TYPE EL5112_Data :
STRUCT
	{attribute addProperty Name "ENC Status Channel 1"}
	ENC_StatusChannel_1 : EL5112_ENC_StatusChannel;
	{attribute addProperty Name "ENC Control Channel 1"}
	ENC_ControlChannel_1 : EL5112_ENC_ControlChannel;
END_STRUCT
END_TYPE

(* stored: Version 1.1.0.1, ProductVersion 3.1.4024.9
   DUT EL5112_Data: Id {85d7b515-701b-0028-322a-39afa7d51a84} *)
